INTERFACE I_V1_127_0_0_1_PackMLPlcStream1_10_00ms EXTENDS I_VirtualInputSource

PROPERTY nV1_TimeLine : ULINT
GET
END_GET
END_PROPERTY

PROPERTY nV1_UnitModeCurrent : DINT
GET
END_GET
END_PROPERTY

END_INTERFACE

(* stored: Itf I_V1_127_0_0_1_PackMLPlcStream1_10_00ms: Id 59950446-618d-4fc8-8e61-7059f82260dd
   Property nV1_TimeLine: Id d9c68758-11e8-461f-bfea-f967f9d612de
   Get Get: Id 9829fd0a-a69b-430b-a12d-766388f294fc
   Property nV1_UnitModeCurrent: Id aaaac9e4-5979-4c3b-a88b-1726f595b429
   Get Get: Id e9579c47-93cf-4d88-a965-008507909a56 *)
